Universal Robots URScript: jelou.script

def initialization():
	global program_counter = 1
end
def main():
	first_trajectory_pose = pose_inv(p[-0.5, -0.3, 0.4, 0.0, 3.14159265358979, 0.0])
	starting_pose_tcp = get_actual_tcp_pose()
	counter = 0
	while(counter < program_counter):
	counter = counter + 1
	end
end
